PROGRAM MAIN
VAR
	// develop branch
	fbReadFile			:FB_ReadFile;
	
    // trigger command execution for OpenWeatherMap samples
    bGetOpenWeatherMap             : BOOL;

    fbHttpClientOpenWeatherMap     : FB_IotHttpClient :=(sHostName:='api.github.com',
                                     bKeepAlive:=TRUE, tConnectionTimeout:=T#10S);

    fbHttpGetOpenWeatherMap        : FB_TestHTTP_Get_openWeatherMap;
END_VAR

//fbReadFile();

// test HTTP GET request
//init client parameters at startup
IF NOT fbHttpClientOpenWeatherMap.bConfigured THEN
    fbHttpClientOpenWeatherMap.nHostPort:= 443;
    fbHttpClientOpenWeatherMap.stTLS.bNoServerCertCheck:= TRUE;
END_IF

IF fbHttpClientOpenWeatherMap.bConfigured THEN
    fbHttpGetOpenWeatherMap(bSend:=bGetOpenWeatherMap, fbClient:=fbHttpClientOpenWeatherMap);
END_IF

fbHttpClientOpenWeatherMap.Execute();

END_PROGRAM

(* stored: Version 1.1.0.1, ProductVersion 3.1.4024.6
   POU MAIN: Id {d70c0d43-1e12-4f89-90c8-3d2f54cc3033}, SpecialFunc None *)
